FUNCTION FIELDBUS_PERCENT_TO_WORD (* Convert a WORD Value Range 0-FAFF to a REAL in the Range 0.0 to 100.0 *)
  (* Standard: SAE J1939; ISO 11783; Description: Copyright (c) 2023 HR Agrartechnik GmbH This program and the accompanying materials are made available under the terms of the Eclipse Public License 2.0 which is available at https://www.eclipse.org/legal/epl-2.0/ SPDX-License-Identifier: EPL-2.0 *)
  (* Version 3.0, 2025-04-14, Patrick Aigner, changed package *)
  (* Version 1.1, 2024-09-19, Franz H??pfinger, HR Agrartechnik GmbH, Update to a more Function like Interface *)
  (* Version 1.0, 2023-10-21, Franz H??pfinger, HR Agrartechnik GmbH *)
  PACKAGE eclipse4diac::signalprocessing;
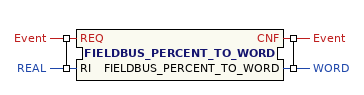
  EVENT_INPUT
    REQ WITH RI;
  END_EVENT
  EVENT_OUTPUT
    CNF WITH FIELDBUS_PERCENT_TO_WORD;
  END_EVENT
  VAR_INPUT
    RI : REAL; (* Input Value *)
  END_VAR
  VAR_OUTPUT
    FIELDBUS_PERCENT_TO_WORD : WORD;
  END_VAR
  BODY IN ST:
PACKAGE signalprocessing;

(* Convert a WORD Value Range 0-FAFF to a REAL in the Range 0.0 to 100.0 *)
FUNCTION FIELDBUS_PERCENT_TO_WORD : WORD
VAR_INPUT
	RI : REAL; // Input Value
END_VAR

FIELDBUS_PERCENT_TO_WORD := UDINT_TO_WORD(REAL_TO_UDINT(RI
	* UDINT_TO_REAL(WORD_TO_UDINT(FIELDBUS_SIGNAL::VALID_SIGNAL_W))));

END_FUNCTION
  END_BODY
END_FUNCTION
